TYPE ST_Event :
STRUCT
	eType:		E_Type;
	eEvent:		E_Event;
	nTimestamp:	ULINT;
	nID:		DINT;
	sMessage:	STRING(255);
	sArguments:	STRING(255);
	sDefault:	STRING(255);
END_STRUCT
END_TYPE

(* stored: Version 1.1.0.1, ProductVersion 3.1.4024.12
   DUT ST_Event: Id {fa6acd16-da1d-4c75-bb6f-6b75cd2ccb39} *)
